RoboDK station: 2E06666VentacPiece_Side1n2n3n4_ivan_2.rdk

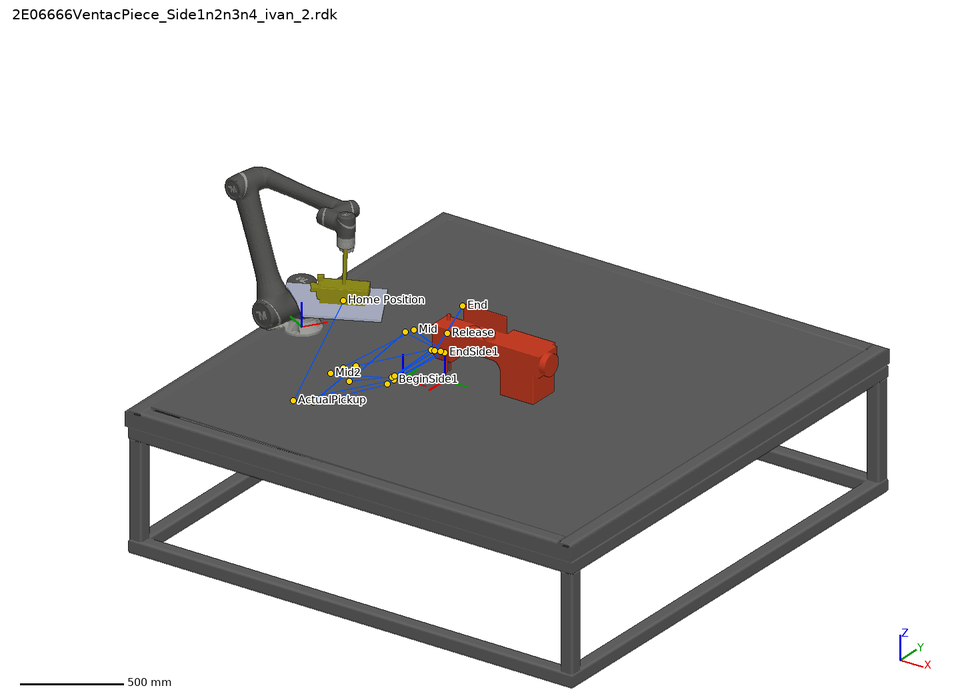
[picture v0: the station drawn from its stored meshes, robots at their saved joint values, targets as dots, program paths as lines]
Station 2E06666VentacPiece_Side1n2n3n4_ivan_2 (saved by RoboDK 5.2.1). Poses are relative to the parent item; angles as X-Y-Z fixed-axis rotations.
Station parameters (name, value as stored): IO_5, 30, OPC-UA, opc.tcp://localhost:4840
  - frame Omron TM12 Base at (190, -120, 780) mm, rotated rx 0 ry 0 rz 60 deg
    - robot Omron TM12: 6 axes, payload 12 kg, reach 1300 mm, repeatability 0.1 mm, weight 33.3 kg
        modified DH rows (alpha deg, a mm, theta deg, d mm): 0, 0, 0, 165.2; 90, 0, 90, 0; 0, 636.1, 0, 0; 0, 557.9, -90, 156.3; -90, 0, 0, 106; 90, 0, 180, 113.15
        base shift (0.29, 0, -5.5) mm
        joint limits [-270, -180, -166, -180, -180, -270] to [270, 180, 166, 180, 180, 270]; home [0, 0, 90, 0, 90, 0]; saved at [-69.04, -19.815, 110.346, 0.067, 87.9, -128.029]
      - tool KVG-gripper, TCP at (0, 0, 285) mm, size 287.4 x 120 x 282 mm, geometry from untitled.obj
        - object 2E06666_REV_C - Copy2 at (18.39, 14.06, 15.2) mm, rotated rx -180 ry 0 rz -91.02 deg, size 361.2 x 491.2 x 12 mm, geometry from 2E06666_REV_C - Copy2.IGS
    - target Home Position (Cartesian target) at (-0.43, -475.84, 354) mm, rotated rx -178.71 ry -1.76 rz 148.98 deg; joints [-69.005, -0.122, 95.32, 175.401, -87.9, 52.005] of Omron TM12
    - target ActualPickup (Cartesian target) at (-403.52, -769.91, 30) mm, rotated rx -179.87 ry 0.95 rz -152 deg; joints [-107.671, 26.496, 96.009, -31.91, 90.757, -225.674] of Omron TM12
    - target BeginSide1 (Cartesian target) at (136.23, -757.31, 25) mm, rotated rx -179.87 ry 0 rz -152.97 deg; joints [-68.109, 18.678, 108.79, -37.593, 90.011, -185.139] of Omron TM12
    - target EndSide1 (Cartesian target) at (483.65, -590.88, 25.16) mm, rotated rx -179.79 ry 0.94 rz -152.97 deg; joints [-39.314, 18.108, 109.711, -38.382, 90.776, -156.339] of Omron TM12
    - target BeginSide2. (Cartesian target) at (143.9, -720.6, 18) mm, rotated rx 178.19 ry 0.77 rz -76.06 deg; joints [-65.537, 16.742, 112.233, -37.888, 88.361, -259.474] of Omron TM12
    - target Mid (Cartesian target) at (447.33, -323.61, 35) mm, rotated rx -179.87 ry 0.95 rz -122.8 deg; joints [-20.127, -0.053, 130.687, -40.967, 90.903, 192.68] of Omron TM12
    - target Mid2 (Cartesian target) at (-119.01, -587.8, 35) mm, rotated rx -179.87 ry 0.95 rz -62.8 deg; joints [-86.187, 4.676, 125.359, -39.11, 89.737, 66.62] of Omron TM12
    - target EndSide2 (Cartesian target) at (445.66, -523.28, 18) mm, rotated rx 178.19 ry 0.77 rz -76.06 deg; joints [-35.922, 13.379, 116.724, -38.347, 89.113, -229.861] of Omron TM12
    - target Mid3 (Cartesian target) at (39.52, -533.02, 18) mm, rotated rx 178.19 ry 0.77 rz -76.06 deg; joints [-67.477, -0.16, 132.808, -41.617, 88.325, -261.414] of Omron TM12
    - target Mid33 (Cartesian target) at (-314.33, -803.28, 18) mm, rotated rx 178.19 ry 0.77 rz 33.94 deg; joints [-101.299, 25.561, 99.565, -36.947, 90.743, -45.24] of Omron TM12
    - target MoveTo3 (Cartesian target) at (-37.22, -553.7, 34.03) mm, rotated rx -179.84 ry 0.65 rz 29.58 deg; joints [-77.014, 17.413, 109.419, 143.138, -89.327, -196.592] of Omron TM12
    - target Start3 (Cartesian target) at (78.52, -806.91, 34.03) mm, rotated rx -179.84 ry 0.65 rz 29.58 deg; joints [-73.009, 38.019, 76.181, 155.816, -89.326, -192.587] of Omron TM12
    - target EndSide3 (Cartesian target) at (468.23, -581.91, 30) mm, rotated rx -179.84 ry 0.65 rz 29.58 deg; joints [-38.814, 16.781, 110.75, -37.138, 89.452, 21.61] of Omron TM12
    - target Side4Switch (Cartesian target) at (399.57, -324.95, 34.03) mm, rotated rx -179.84 ry 0.65 rz 124.58 deg; joints [-21.055, -3.912, 134.502, -41.038, 89.496, -55.635] of Omron TM12
    - target Side4 (Cartesian target) at (-74.15, -698.58, 34.03) mm, rotated rx -179.84 ry 0.65 rz 119.58 deg; joints [-83.288, 12.671, 116.104, -39.44, 90.104, -112.866] of Omron TM12
    - target BeginSide4 (Cartesian target) at (148.41, -739.92, 34.03) mm, rotated rx -179.84 ry 0.65 rz 119.58 deg; joints [-66.677, 16.766, 110.503, -37.937, 89.909, -96.255] of Omron TM12
    - target EndSide4 (Cartesian target) at (442.86, -569.92, 34.03) mm, rotated rx -179.84 ry 0.65 rz 119.58 deg; joints [-39.441, 14.179, 114.058, -38.789, 89.614, -69.021] of Omron TM12
    - target Release (Cartesian target) at (576.89, -422.07, 34.03) mm, rotated rx -179.84 ry 0.65 rz 119.58 deg; joints [-23.27, 29.808, 90.162, 149.606, -89.475, 127.15] of Omron TM12
    - target End (Cartesian target) at (772.86, -179.92, 34.03) mm, rotated rx -179.84 ry 0.65 rz 119.58 deg; joints [-1.416, 19.913, 105.84, -35.95, 89.355, -30.995] of Omron TM12
  - frame Tool at (0, 1000, 0) mm
    - object Machine at (1443.88, -1066.05, 820) mm, rotated rx 0 ry 0 rz -90 deg, size 180 x 665 x 356.6 mm, geometry from Machine.IGS
  - object Table 108x114x32 IN at (0, 0, 0) mm, size 2628.9 x 2679.7 x 778.4 mm, geometry from Table-108x114x32-IN.sld
  - program Prog1 (29 instructions, listed below)
  - frame Needle at (1090, -200, 780) mm, rotated rx 0 ry 0 rz -90 deg
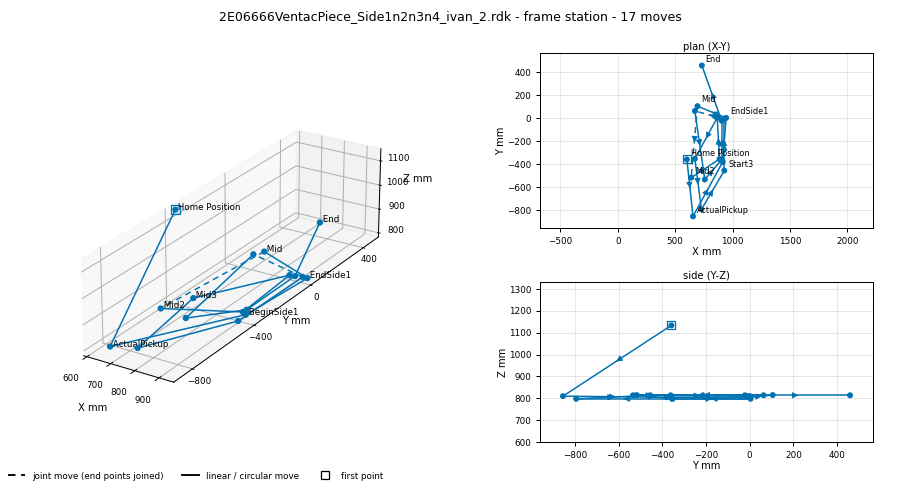
[picture p0: tool path of 2E06666VentacPiece_Side1n2n3n4_ivan_2.rdk in frame station, 17 of 17 moves have a stored position in this frame; points joined in program order, loops and branches not executed]

--- program Prog1 (robot Omron TM12) ---
  Set Ref.: Omron TM12 Base
  Set Tool: KVG-gripper
  Accurate (rounding -1 mm)
  MoveL (Home Position)
  MoveL (ActualPickup)
  Set IO_5=40
  MoveL (BeginSide1)
  Set IO_5=20
  MoveL (EndSide1)
  Set IO_5=30
  MoveL (Mid)
  MoveJ (Mid2)
  MoveL (BeginSide2.)
  Set IO_5=20
  MoveL (EndSide2)
  Set IO_5=30
  MoveL (Target 28) -> target Mid3
  MoveL (Target 27) -> target Mid33
  MoveL (Start3)
  Set IO_5=20
  MoveL (EndSide3)
  Set IO_5=30
  MoveJ (Side4Switch)
  MoveL (Side4)
  MoveL (BeginSide4)
  Set IO_5=20
  MoveL (EndSide4)
  Set IO_5=30
  MoveL (End)
